Fanuc KAREL source: kt00401.KL

-- PROVISIONAL review KL for V1013-1; original PC SHA256 049ea0cfa262c239f4d991f34e1f751580a45e062d6e3a11d69e4f6688868017
-- Incomplete behavior may be omitted. Consult companion uncertainty JSON. Do not deploy.
PROGRAM KT00401
%NOLOCKGROUP
VAR
  I1 : INTEGER
  I2 : INTEGER
  OUT : BOOLEAN
BEGIN
  -- UNRESOLVED_PC offsets 5-16; opcodes 2E,23
  -- UNRESOLVED_PC offsets 21-32; opcodes 2E,23
  -- UNRESOLVED_PC offsets 37-48; opcodes 2E,23
  -- UNRESOLVED_PC offsets 53-64; opcodes 2E,23
  -- UNRESOLVED_PC offsets 69-88; opcodes 21,21,5B,23
  -- UNRESOLVED_PC offsets 93-97; opcodes 7F
END KT00401
